// TIA Portal project "Project3" (V16)

(* hardware
DEVICE "S7-1200 station_1"  S7-1200 Station
   slot 0: "Rack_0"  S7-1200 Rack  Rack  V1.0
   slot 1: "PLC_1"  CPU 1215C DC/DC/DC  6ES7 215-1AG40-0XB0  V4.4
*)

// ===== PLC "PLC_1"  CPU 1215C DC/DC/DC =====

VAR_GLOBAL   // PLC tag table "Default tag table"
   "Tag_2" AT %Q0.2 : Bool;
   "Tag_1" AT %M1.0 : Bool;
   "Tag_3" AT %I0.1 : Bool;
   "Tag_4" AT %I0.0 : Bool;
   "Start" AT %M0.0 : Bool;
   "Tag_6" AT %M0.1 : Bool;
   "Axis_1_Pulse" AT %Q0.0 : Bool;
   "Axis_2_Pulse" AT %Q0.1 : Bool;
   "Axis_2_Direction" AT %Q0.6 : Bool;
   "Axis_1_Direction" AT %Q0.4 : Bool;
   "Axis_2_Direction(1)" AT %Q0.5 : Bool;
   "Tag_7" AT %M0.7 : Bool;
   "Tag_8" AT %M0.6 : Bool;
   "Tag_9" AT %M0.5 : Bool;
   "Tag_10" AT %M0.4 : Bool;
   "Tag_11" AT %M0.3 : Bool;
   "Tag_12" AT %M0.2 : Bool;
   "Finish" AT %Q1.0 : Bool;
   "Xilanh" AT %Q1.1 : Bool;
END_VAR

DATA_BLOCK "Data_block_1"   // DB1
{ S7_Optimized_Access := 'FALSE' }
VERSION : 0.1
   VAR
      x : Real;
      y : Real;
      z : Real;
      m1 : Real;
   END_VAR
BEGIN
END_DATA_BLOCK

// folder: System blocks/Program resources

DATA_BLOCK "IEC_Timer_0_DB_1"   // DB15
{ S7_Optimized_Access := 'TRUE' }
AUTHOR : Simatic
FAMILY : IEC
NAME : IEC_TMR
VERSION : 1.0
// stored: InstanceOfName IEC_TIMER
"IEC_TIMER"
BEGIN
END_DATA_BLOCK

// folder: (top level)

DATA_BLOCK "Axis_1"   // DB2, Motion_DB
{ S7_Optimized_Access := 'TRUE' }
AUTHOR : SIMATIC
FAMILY : BasicMC
NAME : TO_PosAx
VERSION : 7.0
// stored: InstanceOfName TO_PositioningAxis
"TO_PositioningAxis"
BEGIN
   // Axis.DirectionOutputEnabledCU = TRUE
   // Axis.OnlinePtoModeCU = 16#0000_0002
   // Axis.SelectedChannel2EnumCU = %Q0.4
   // Axis.SelectedChannel1EnumCU = %Q0.0
   // Pulse.MinDeltaDeltaFrequencyCU = 0.004
   // Pulse.MaxDeltaDeltaFrequencyCU = 1.0E+10
   // Pulse.MinDeltaFrequencyCU = 0.005
   // Pulse.MaxDeltaFrequencyCU = 9.5E+9
   // Pulse.MinFrequencyCU = 1.0
   // Pulse.MaxFrequencyCU = 100000.0
   // Pulse.OutputSourceCU = 16#0000_0000
   // Axis.SelectPTO = 0
END_DATA_BLOCK

DATA_BLOCK "Axis_2"   // DB3, Motion_DB
{ S7_Optimized_Access := 'TRUE' }
AUTHOR : SIMATIC
FAMILY : BasicMC
NAME : TO_PosAx
VERSION : 7.0
// stored: InstanceOfName TO_PositioningAxis
"TO_PositioningAxis"
BEGIN
   // Axis.DirectionOutputEnabledCU = TRUE
   // Axis.OnlinePtoModeCU = 16#0000_0002
   // Axis.SelectedChannel2EnumCU = %Q0.5
   // Axis.SelectedChannel1EnumCU = %Q0.1
   // Pulse.MinDeltaDeltaFrequencyCU = 0.004
   // Pulse.MaxDeltaDeltaFrequencyCU = 1.0E+10
   // Pulse.MinDeltaFrequencyCU = 0.005
   // Pulse.MaxDeltaFrequencyCU = 9.5E+9
   // Pulse.MinFrequencyCU = 1.0
   // Pulse.MaxFrequencyCU = 100000.0
   // Pulse.OutputSourceCU = 16#0000_0000
   // Axis.SelectPTO = 1
   // Axis.OnlinePtoIndexCU = 1
END_DATA_BLOCK

DATA_BLOCK "Axis_3"   // DB4, Motion_DB
{ S7_Optimized_Access := 'TRUE' }
AUTHOR : SIMATIC
FAMILY : BasicMC
NAME : TO_PosAx
VERSION : 7.0
// stored: InstanceOfName TO_PositioningAxis
"TO_PositioningAxis"
BEGIN
   // Axis.DirectionOutputEnabledCU = TRUE
   // Axis.OnlinePtoModeCU = 16#0000_0002
   // Axis.SelectedChannel2EnumCU = %Q0.6
   // Axis.SelectedChannel1EnumCU = %Q0.2
   // Pulse.MinDeltaDeltaFrequencyCU = 0.004
   // Pulse.MaxDeltaDeltaFrequencyCU = 1.0E+10
   // Pulse.MinDeltaFrequencyCU = 0.005
   // Pulse.MaxDeltaFrequencyCU = 9.5E+9
   // Pulse.MinFrequencyCU = 1.0
   // Pulse.MaxFrequencyCU = 100000.0
   // Pulse.OutputSourceCU = 16#0000_0000
   // Axis.SelectPTO = 2
   // Axis.OnlinePtoIndexCU = 2
END_DATA_BLOCK

ORGANIZATION_BLOCK "Main"   // OB1, LAD, ProgramCycle
TITLE = "Main Program Sweep (Cycle)"
{ S7_Optimized_Access := 'TRUE' }
VERSION : 0.1
   VAR_INPUT
      Initial_Call : Bool;   // Initial call of this OB
      Remanence : Bool;   // =True, if remanent data are available
   END_VAR
BEGIN

REGION Network 1: AXIS X
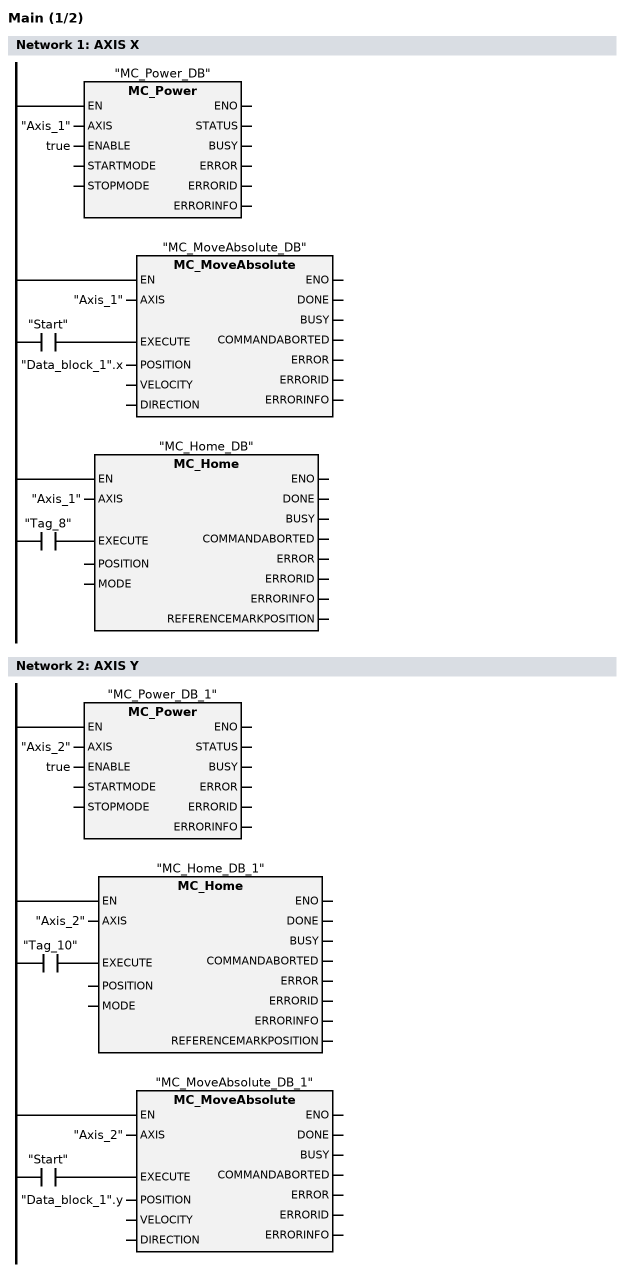
   "MC_Power_DB"(Axis := "Axis_1", Enable := true);   // MC_Power
   "MC_MoveAbsolute_DB"(Axis := "Axis_1", Execute := "Start", Position := "Data_block_1".x);   // MC_MoveAbsolute
   "MC_Home_DB"(Axis := "Axis_1", Execute := "Tag_8");   // MC_Home
END_REGION

REGION Network 2: AXIS Y
   "MC_Power_DB_1"(Axis := "Axis_2", Enable := true);   // MC_Power
   "MC_Home_DB_1"(Axis := "Axis_2", Execute := "Tag_10");   // MC_Home
   "MC_MoveAbsolute_DB_1"(Axis := "Axis_2", Execute := "Start", Position := "Data_block_1".y);   // MC_MoveAbsolute
END_REGION

REGION Network 3: AXIS Z
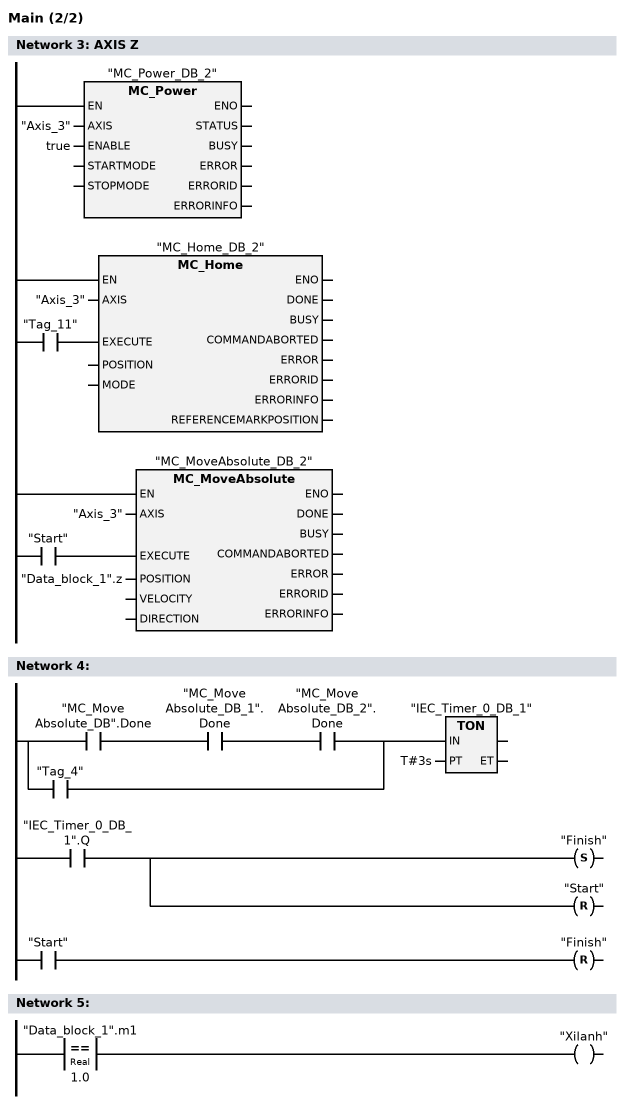
   "MC_Power_DB_2"(Axis := "Axis_3", Enable := true);   // MC_Power
   "MC_Home_DB_2"(Axis := "Axis_3", Execute := "Tag_11");   // MC_Home
   "MC_MoveAbsolute_DB_2"(Axis := "Axis_3", Execute := "Start", Position := "Data_block_1".z);   // MC_MoveAbsolute
END_REGION

REGION Network 4
   "IEC_Timer_0_DB_1".TON(IN := ("MC_MoveAbsolute_DB".Done AND "MC_MoveAbsolute_DB_1".Done AND "MC_MoveAbsolute_DB_2".Done) OR "Tag_4",
                          PT := T#3s);
   IF "IEC_Timer_0_DB_1".Q THEN
       "Finish" := TRUE;
       "Start" := FALSE;
   END_IF;
   IF "Start" THEN "Finish" := FALSE; END_IF;
END_REGION

REGION Network 5
   RUNG wire#powerrail
      { S7_Templates := "SrcType := Real" } EQ_Contact(in1 := "Data_block_1".m1, in2 := 1.0)
      Coil( "Xilanh" )
   END_RUNG
   // the same network as SCL:
   "Xilanh" := "Data_block_1".m1 = 1.0;
END_REGION
END_ORGANIZATION_BLOCK